(* IEC 61131-3 sources: generating_plc_code_with_llms/Code#2/CodeLlama/third run, 21 files *)

(* ---- 10.st ---- *)
// 23.59233784675598s
// 2
```
FUNCTION SIGMOID(X : REAL) : REAL;
VAR
    Y : REAL;
BEGIN
    IF (X < 0.0) THEN
        Y := 1.0 / (1.0 + EXP(-X));
    ELSE
        Y := X;
    END_IF;
    RETURN Y;
END_FUNCTION;
```

(* ---- 11.st ---- *)
// 22.66158437728882s
// 2
```
FUNCTION sign(x:REAL):REAL;
VAR
    y:REAL;
BEGIN
    IF (x > 0) THEN
        y := 1;
    ELSIF (x < 0) THEN
        y := -1;
    ELSE
        y := 0;
    END_IF;
    RETURN y;
END_FUNCTION;
```

(* ---- 12.st ---- *)
// 19.898288249969482s
// 2
```
FUNCTION SINH(X:REAL):REAL;
VAR
    EXP_X : REAL;
BEGIN
    EXP_X := EXP(X);
    RETURN (EXP_X - 1/EXP_X)/2;
END_FUNCTION;
```

(* ---- 13.st ---- *)
// 36.65593123435974s
// 2
```
FUNCTION SelectNumber(nNumber : INT) : BOOL;
VAR
    bFound : BOOL := FALSE;
END_VAR

bFound := FALSE;
REPEAT
    IF aNumbers[nCnt] = nNumber THEN
        bFound := TRUE;
        EXIT;
    END_IF;
    nCnt := nCnt + 1;
UNTIL (nCnt > MAXNUMBERS) OR bFound;

IF nCnt > MAXNUMBERS THEN
    RETURN FALSE;
ELSE
    RETURN TRUE;
END_IF;
END_FUNCTION;
```

(* ---- 14.st ---- *)
// 51.47999310493469s
// 3
```
FUNCTION FC1001 :BOOL
VAR_INPUT
	MEW: REAL;
	SP: REAL;
	HYS: REAL;
END_VAR
VAR_IN_OUT
 	OUT:BOOL;
END_VAR
VAR
 	P_HYS: REAL;
END_VAR
BEGIN
	IF (MEW > SP) THEN
		IF (MEW - SP > HYS * SP) THEN
			OUT := TRUE;
		ELSE
			OUT := FALSE;
		END_IF;
	ELSIF (MEW < SP) THEN
		IF (SP - MEW > HYS * SP) THEN
			OUT := TRUE;
		ELSE
			OUT := FALSE;
		END_IF;
	ELSE
		OUT := FALSE;
	END_IF;
END_FUNCTION
```

(* ---- 15.st ---- *)
// 49.1918363571167s
// 2
```
FUNCTION FC1002 :BOOL
VAR_INPUT
	E_A, SENSOR: BOOL;
	ZEITW: TIME;
END_VAR
VAR_IN_OUT
	ZEIT:TON;
	P_HU, P_AL: BOOL;
END_VAR
BEGIN
	IF E_A THEN
		IF SENSOR THEN
			P_HU := TRUE;
			ZEIT := ZEITW;
		ELSE
			IF (ZEITW - ZEIT) > T#3s THEN
				P_AL := TRUE;
				P_HU := FALSE;
			END_IF;
		END_IF;
	END_IF;
END_FUNCTION;
```

(* ---- 17.st ---- *)
// 47.26889777183533s
// 4
```
FUNCTION TEXT_OUTPUT
VAR
    iTemp : INT;
    iHumidity : INT;
    sShowText : STRING[80];
END_VAR

IF (aiOutside < 18) THEN
    sShowText := 'Cold';
ELSIF (aiOutside >= 18 AND aiOutside <= 25) THEN
    IF (aiHumidity >= 40 AND aiHumidity <= 75) THEN
        sShowText := 'Opt';
    ELSE
        sShowText := 'Temp. OK';
    END_IF;
ELSE
    sShowText := 'Hot';
END_IF;

sShowText;
END_FUNCTION;
```

(* ---- 18.st ---- *)
// 50.14126205444336s
// 2
```
FUNCTION FC1003 : VOID
VAR_INPUT
    IN_R:REAL;
    IN_MAX, IN_MIN:REAL;
    OUT_MAX, OUT_MIN:REAL;
END_VAR
VAR_OUTPUT
    OUT_R:REAL;
    FEH:BOOL;
END_VAR
VAR_TEMP
    DIFF1, DIFF2:REAL;
END_VAR
BEGIN
    IF IN_MAX = IN_MIN THEN
        FEH := FALSE;
        OUT_R := 0.0;
    ELSE
        DIFF1 := (IN_MAX - IN_MIN) / 255.0;
        DIFF2 := (OUT_MAX - OUT_MIN) / (IN_MAX - IN_MIN);
        IF IN_R < IN_MIN THEN
            FEH := FALSE;
            OUT_R := OUT_MIN;
        ELSEIF IN_R > IN_MAX THEN
            FEH := FALSE;
            OUT_R := OUT_MAX;
        ELSE
            FEH := TRUE;
            OUT_R := OUT_MIN + DIFF2 * (IN_R - IN_MIN);
        END_IF;
    END_IF;
END_FUNCTION
```

(* ---- 2.st ---- *)
// 25.620573043823242s
// 2
```
FUNCTION binomial(N : INT; K : INT) : INT;
VAR
    result : INT := 1;
    i : INT := 0;
END_VAR
WHILE (i <= N - K) DO
    result := result * (N - i);
    i := i + 1;
END_WHILE;
result := result / factorial(K);
RETURN result;
END_FUNCTION;
```

(* ---- 3.st ---- *)
// 28.61563515663147s
// 2
```
FUNCTION Fibunacci(X: INT): INT
BEGIN
    IF (X = 0) THEN
        RETURN 0;
    ELSEIF (X = 1) THEN
        RETURN 1;
    ELSE
        t1 := Fibunacci(X - 2);
        t2 := Fibunacci(X - 1);
        x_tmp := t1 + t2;
        RETURN x_tmp;
    END_IF;
END_FUNCTION
```

(* ---- 8.st ---- *)
// 57.669310569763184s
// 2
```
FUNCTION LambertW(X : REAL) : REAL
VAR
    w : REAL;
    i : INT;
    we : REAL;
    w1e : REAL;
    ewx : REAL;
    last : DWORD;
END_VAR
BEGIN
    IF X < 0 THEN
        RETURN -1;
    END_IF;
    i := 0;
    we := 1;
    w1e := 1;
    ewx := 1;
    last := 0;
    WHILE (i < 20) AND (ABS(w - w1e) > 1E-6) DO
        i := i + 1;
        we := we * X / (i * (i + 1));
        w1e := w1e + we;
        ewx := ewx * ABS(X);
        IF last = 0 THEN
            last := ABS(w - w1e) / ewx;
        ELSE
            last := ABS(last - (ABS(w - w1e) / ewx));
        END_IF;
    END_WHILE;
    RETURN w1e;
END_FUNCTION;
```

(* ---- 9.st ---- *)
// 24.359095573425293s
// 2
```
FUNCTION ISLEAPYEAR(YEAR : INT) : BOOL;
BEGIN_ISLEAPYEAR
    IF (YEAR MOD 4 = 0 AND YEAR MOD 100 <> 0) OR YEAR MOD 400 = 0 THEN
        RETURN TRUE;
    ELSE
        RETURN FALSE;
    END_IF;
END_ISLEAPYEAR;
```

(* ---- 19.st ---- *)
// 71.44161653518677s
// 3
```
FUNCTION_BLOCK FB1005
VAR_INPUT
    START:BOOL;
    DICKE, V_MAX, V_MIN:REAL;
END_VAR
VAR_OUTPUT
    D_MAX, D_MIN:REAL;
    P1:BOOL;
END_VAR
VAR
    FO:BOOL;
END_VAR
PROGRAM
    IF START THEN
        FO := TRUE;
        D_MAX := 0.0;
        D_MIN := 0.0;
    END_IF;
    IF FO AND NOT(START) THEN
        IF DICKE > V_MAX OR DICKE < V_MIN THEN
            P1 := TRUE;
        ELSE
            P1 := FALSE;
        END_IF;
        IF DICKE > D_MAX THEN
            D_MAX := DICKE;
        END_IF;
        IF DICKE < D_MIN THEN
            D_MIN := DICKE;
        END_IF;
    END_IF;
END_PROGRAM
```

(* ---- 20.st ---- *)
// 82.86100125312805s
// 2
```
FUNCTION_BLOCK INTERLOCK
VAR_INPUT
    I1 : BOOL;
    I2 : BOOL;
    TL : TIME;
END_VAR
VAR_OUTPUT
    Q1 : BOOL;
    Q2 : BOOL;
END_VAR
VAR
    T1 : TOF;
    T2 : TOF;
END_VAR

PROGRAM INTERLOCK
VAR
    I1 : BOOL := FALSE;
    I2 : BOOL := FALSE;
    TL : TIME := '0:0:0.5';
    Q1 : BOOL;
    Q2 : BOOL;
END_VAR

IF (I1) THEN
    IF (NOT(T1)) THEN
        Q1 := TRUE;
        T1 := TOF;
    END_IF;
ELSIF (I2) THEN
    IF (NOT(T2)) THEN
        Q2 := TRUE;
        T2 := TOF;
    END_IF;
END_IF;

IF (Q1 AND NOT(Q2)) OR (Q2 AND NOT(Q1)) THEN
    IF ((I1 AND NOT(T1)) OR (I2 AND NOT(T2))) THEN
        Q1 := TRUE;
        T1 := TOF;
    END_IF;
ELSE
    Q1 := FALSE;
END_IF;

IF (Q2 AND NOT(Q1)) THEN
    IF ((I1 AND NOT(T1)) OR (I2 AND NOT(T2))) THEN
        Q2 := TRUE;
        T2 := TOF;
    END_IF;
ELSE
    Q2 := FALSE;
END_IF;

END_PROGRAM
```

(* ---- 21.st ---- *)
// 435.3805413246155s
// 2
```
FUNCTION_BLOCK BURNER
VAR_INPUT
    IN : BOOL;
    STAGE2 : BOOL;
    OVER_TEMP : BOOL;
    OIL_TEMP : BOOL := TRUE;
    FLAME : BOOL;
    RST : BOOL;
    RST_TIMER : BOOL;
    PRE_HEAT_TIME : TIME := t#5s;
    PRE_VENT_TIME : TIME := t#15s;
    PRE_IGNITE_TIME : TIME := t#15s;
    POST_IGNITE_TIME : TIME := t#25s;
    STAGE2_DELAY : TIME := t#10s;
    SAFETY_TIME : TIME := t#5s;
    LOCKOUT_TIME : TIME := t#10s;
    MULTIPLE_IGNITION : BOOL := TRUE;
    KW1 : REAL;
    KW2 : REAL;
END_VAR
VAR_OUTPUT
    MOTOR : BOOL;
    COIL1 : BOOL;
    COIL2 : BOOL;
    PRE_HEAT : BOOL;
    IGNITE : BOOL;
    FAIL : BOOL;
    KWH : REAL;
    STATUS : BYTE;
END_VAR
VAR_IN_OUT
    RUNTIME1 : UDINT;
    RUNTIME2 : UDINT;
    CYCLES : UDINT;
END_VAR
VAR
    state : INT;
    last : TIME;
    tx : TIME;
    last_change : TIME;
    timer1 : TON;
    timer2 : TON;
    oil_temp_last : BOOL;
    cycles2 : UDINT;
END_VAR

IF IN THEN
    IF NOT OVER_TEMP THEN
        IF NOT FLAME THEN
            IF NOT RST THEN
                IF NOT RST_TIMER THEN
                    state := 110;
                    last := TIME;
                    tx := PRE_HEAT_TIME;
                    timer1.PT := PRE_HEAT_TIME;
                    timer2.PT := STAGE2_DELAY;
                    IF NOT OIL_TEMP THEN
                        oil_temp_last := FALSE;
                    ELSE
                        oil_temp_last := TRUE;
                    END_IF;
                ELSE
                    state := 113;
                    last := TIME;
                    tx := STAGE2_DELAY;
                    timer1.PT := PRE_HEAT_TIME;
                     _TIME;
                      ;

                 0_TIME;
                                                                                                                                                                                                                                                    TIME;
                                                                                                                                                                                                                                                                                                     _TIME;
                                                                                                                                      ;

                 0_TIME;
                                                                                                                                                                                                    TIME;

                    TIME;
                                                                                                                                                     _TIME;
                                                                                                                                                                                      ;

                 0_TIME;
                                                                                                                                                                                                                                                                                                                                                    TIME;
                                                                                                                                                     _TIME;
                                                                                                                                                                                                                                                      ;
                 0_TIME;

                    TIME;
                                                                                                                                                     _TIME;
                                                                                                                                                                                                                                                      ;
                 0_TIME;

                                                                                                                                                                                                                                                    TIME;
                                                                                                                                                     _TIME;
                                                                                                                                                                                                                                                      ;
                 0_TIME;

                                                                                                                                                                                                                                                    TIME;
                                                                                                                                                     _TIME;

                    ;
                 0_TIME;

                                                                                                                                                                                                                                    TIME;
                                                                                                                                     _TIME;

                    ;
                 0_TIME;

                                                      _TIME;

                                                                                                                                                                                                                                                                                                                     TIME;
                    _TIME;
                                                                                                                                                                                                                                                 0_TIME;
                                                                                                      ;

                                                                                                                                                                                                                                                                                                                     TIME;
                    _TIME;
                                                                                                                                                                                                                                                 0_TIME;
                                                                                                                                      ;

                        TIME;
                                                                                                                                                                                                                     _TIME;

                                                                 0_TIME;
                                                                                                                                      ;

                                                                                                                                                                                                                                                                                                                     _TIME;
                                                                                                        TIME;
                                                                    TIME;
                 0_TIME;
                                                                                                                                    ;
                                      _TIME;

                                                                                                                                                                                                                                                                                                                                                                                                 0_TIME;
                                                                                                                                    TIME;
                                                                                                   ;
                                                                                                      _TIME;

                                                                                                                                 0_TIME;
                                                                                                                                                                                    TIME;
                                                   ;
                                                                                                      _TIME;

                 0_TIME;
                                                                                                                                                                                                                                                                                                   ;
                     _TIME;
                      TIME;

                                                                                                                                                                                                                 0_TIME;
                                                                                                                                                                                                                                                                                                   ;
                     _TIME;
                    TIME;

                    _TIME;
                                                 0_TIME;

                    TIME;
                                                                                                                                                   ;

                                                                                                                                                                                                                                                                                                                                                    _TIME;
                 0_TIME;
                    TIME;

                                                                                   ;

                    TIME;

                                                                                                                                                                                                                                                                                                                 0_TIME;
                                                                                                                                                                                                                                   ;
                     _TIME;
                                                                                                                                                    TIME;
                    ;

                                                                                                                                                                                                                                                 0_TIME;
                                                                                                                        TIME;

                                     _TIME;

                                                                                                                      ;

                                                                                                                                                                                 0_TIME;

                     _TIME;
                                                                                                                                                                                                                                                                                                      ;
                    TIME;

                 0_TIME;

(* ---- 1.st ---- *)
// 43.99788689613342s
// 2
```
PROGRAM Alarms
VAR
	xAllOn : BOOL;
	xAllOff : BOOL;

	xAlarm1 : BOOL;
    xAlarm2 : BOOL;
END_VAR

FUNCTION Alarm(xAlarm : BOOL) : BOOL
VAR
	xAlarm : BOOL;
END_VAR
RETURN xAlarm;
END_FUNCTION

PROGRAM
BEGIN
	IF (xAllOn) THEN
		xAlarm1 := TRUE;
		xAlarm2 := TRUE;
	ELSIF (xAllOff) THEN
		xAlarm1 := FALSE;
		xAlarm2 := FALSE;
	END_IF;
END_PROGRAM
```

(* ---- 16.st ---- *)
// 35.92371940612793s
// 2
```
PROGRAM TrafficLight
VAR
    North_green : BOOL;
    North_yellow : BOOL;
    North_red : BOOL;
    East_green : BOOL;
    East_yellow : BOOL;
    East_red : BOOL;
    T1 : TON;
END_VAR

IF (T1 < 5000) THEN
    North_green := TRUE;
    East_red := TRUE;
ELSIF (T1 >= 5000 AND T1 < 6000) THEN
    North_yellow := TRUE;
    East_red := TRUE;
ELSIF (T1 >= 9500 AND T1 < 10000) THEN
    North_red := TRUE;
    East_green := TRUE;
ELSE
    North_red := TRUE;
    East_yellow := TRUE;
END_IF;
END_PROGRAM;
```

(* ---- 4.st ---- *)
// 52.24701428413391s
// 2
```
PROGRAM fillLevelCheck
VAR
    aiLevel : INT;
    PercentLevel : UINT;
    doLow : BOOL;
    doOk : BOOL;
    doHigh : BOOL;
    doAlarm : BOOL;
END_VAR

CASE aiLevel OF
    0..10: doLow := TRUE; doOk := FALSE; doHigh := FALSE;
    11..30: doLow := FALSE; doOk := TRUE; doHigh := FALSE;
    ELSE: doLow := FALSE; doOk := FALSE; doHigh := TRUE;
END_CASE

IF PercentLevel < 1 THEN
    doAlarm := TRUE;
END_IF

IF doLow THEN
    OUTPUT('LOW');
ELSIF doOk THEN
    OUTPUT('OK');
ELSIF doHigh THEN
    OUTPUT('HIGH');
ELSE
    OUTPUT('ALARM');
END_IF

END_PROGRAM
```

(* ---- 5.st ---- *)
// 81.71327662467957s
// 2
```
PROGRAM GATE_CONTROLLER
VAR
    Start_Loop : BOOL := FALSE;
    one_hour : TIME := T#1h;
    One_Hour_Timer : TON;
    Gate_Open : BOOL := FALSE;
    Close_Gate_Inst : BOOL := FALSE;
    Sensed_Car : BOOL := FALSE;
    Sensed_Car_Inst : BOOL := FALSE;
    Sensed_App : BOOL := FALSE;
    Mobile_Inst : BOOL := FALSE;
    Auth : STRING;
    my_defined_str : STRING := 'abcd';
END_VAR

IF Start_Loop THEN
    One_Hour_Timer.TON := TRUE;
ELSE
    IF One_Hour_Timer.Q THEN
        IF Gate_Open THEN
            Close_Gate_Inst := TRUE;
        ELSE
            IF Sensed_Car OR Sensed_App THEN
                IF Auth = my_defined_str THEN
                    Gate_Open := TRUE;
                END_IF;
            END_IF;
        END_IF;
    END_IF;
END_IF;

IF Close_Gate_Inst THEN
    Gate_Open := FALSE;
END_IF;

IF Sensed_Car OR Sensed_App THEN
    IF Auth = my_defined_str THEN
        Mobile_Inst := TRUE;
    END_IF;
END_IF;

IF Mobile_Inst THEN
    IF NOT Gate_Open THEN
        Gate_Open := TRUE;
    ELSE
        Close_Gate_Inst := TRUE;
    END_IF;
END_IF;
```

(* ---- 6.st ---- *)
// 119.65785598754883s
// 2
```
PROGRAM CraneLift
VAR
    WAIT : UINT:= 0;
    TOP_POSITION : UINT:= 1;
    BOTTOM_POSITION : UINT:= 2;
    GETBOX : UINT:= 3;
    UNLOAD_POSITION : UINT:= 4;
    UNLOAD_BOX : UINT:= 5;
END_VAR

VAR
    (*-- digital outputs*)
    doConvTop: BOOL;
    doConvBottom: BOOL;
    doConvLift: BOOL;
    doLiftTop: BOOL;
    doLiftBottom: BOOL;
    doLiftUnload: BOOL;
    (*-- digital inputs*)
    diConvTop: BOOL;
    diConvBottom: BOOL;
    diLiftTop: BOOL;
    diLiftBottom: BOOL;
    diLiftUnload: BOOL;
    diBoxLift: BOOL;
    (*-- status variables*)
    selectLift: UINT;
    ConvTopOn: BOOL;
    ConvBottomOn: BOOL;
END_VAR

PROGRAM
    IF (diConvTop) THEN
        doConvTop := TRUE;
        ConvTopOn := TRUE;
    END_IF;
    IF (diConvBottom) THEN
        doConvBottom := TRUE;
        ConvBottomOn := TRUE;
    END_IF;
    IF (diLiftTop) THEN
        doLiftTop := TRUE;
    END_IF;
    IF (diLiftBottom) THEN
        doLiftBottom := TRUE;
    END_IF;
    IF (diBoxLift) THEN
        doConvLift := TRUE;
    END_IF;
    IF (doConvTop AND ConvTopOn) THEN
        selectLift := TOP_POSITION;
    ELSIF (doConvBottom AND ConvBottomOn) THEN
        selectLift := BOTTOM_POSITION;
    ELSE
        selectLift := GETBOX;
    END_IF;
    IF (selectLift = GET

(* ---- 7.st ---- *)
// 62.37231373786926s
// 2
```
PROGRAM PLC_Crane
VAR
    MAX_INDEX: USINT := 4;
END_VAR
VAR
    aWeights : ARRAY[0..MAX_INDEX] OF INT;
    iCnt : USINT;
    sumWeight : DINT;
    avgWeight : INT;
END_VAR
FUNCTION GetWeight(iIndex: USINT) : INT
VAR
    iWeight : INT;
END_VAR
iWeight := aWeights[iIndex];
RETURN iWeight;
END_FUNCTION
PROGRAM
aWeights[0] := 12345;
aWeights[1] := 23456;
aWeights[2] := 34567;
aWeights[3] := 45678;
iCnt := 0;
sumWeight := 0;
WHILE iCnt < MAX_INDEX DO
    sumWeight := sumWeight + GetWeight(iCnt);
    iCnt := iCnt + 1;
END_WHILE
avgWeight := sumWeight / MAX_INDEX;
ENDPROGRAM
```
